// TwinCAT 3 PLC project lev_fsm
// ProgramVersion: 3.1.4023.0
// libraries:
//   Tc2_SerialCom, * (Beckhoff Automation GmbH)
//   Tc2_Standard, * (Beckhoff Automation GmbH)
//   Tc2_System, * (Beckhoff Automation GmbH)
//   Tc2_Utilities, * (Beckhoff Automation GmbH)
//   Tc3_Module, * (Beckhoff Automation GmbH)
// project tree:
//   DUTs/ E_FsmError.TcDUT (not stored), E_FsmState.TcDUT (not stored), mag_bus.TcDUT, ST_Event.TcDUT (not stored), sus_bus.TcDUT (not stored)
//   / PlcTask.TcTTO (not stored)
//   POUs/ getFmagnetic.TcPOU, getTrajectory.TcPOU (not stored), LevitationEqualizingController.TcPOU, MAIN.TcPOU (not stored), runIpcFsm.TcPOU (not stored)
//   POUs/nicht aufgerufen/ FiniteStateMachine.TcPOU, GenerateTrajectory.TcPOU (not stored), Trajectory.TcPOU, UpdateEventTimestampWithSystemTime.TcPOU

// ---- DUTs/mag_bus.TcDUT
TYPE mag_bus:
    STRUCT
        Fmat: ARRAY [0..143] OF LREAL;
        zmat: ARRAY [0..143] OF LREAL;
        invFmat: ARRAY [0..143] OF LREAL;
        F_grid: ARRAY [0..16383] OF LREAL;
        z_grid: ARRAY [0..16383] OF LREAL;
        i_grid: ARRAY [0..16383] OF LREAL;
    END_STRUCT
END_TYPE

// ---- POUs/getFmagnetic.TcPOU
FUNCTION getFmagnetic : LREAL
VAR_INPUT
    I: LREAL;
    z: LREAL;
END_VAR
VAR
    Fmag_tmp: LREAL;
    Fmag_tmp_0: LREAL;
    Fmag_tmp_1: LREAL;
    Fmag_tmp_2: LREAL;
    Fmag_tmp_3: LREAL;
    Fmag_tmp_4: LREAL;
END_VAR

(* MATLAB Function: '<Root>/getFmag' *)
(* MATLAB Function 'getFmag': '<S1>:1' *)
(* '<S1>:1:2' p00 =  -4.108e+05; *)
(* '<S1>:1:3' p10 =        3267; *)
(* '<S1>:1:4' p01 =   1.697e+05; *)
(* '<S1>:1:5' p20 =       61.45; *)
(* '<S1>:1:6' p11 =       -1147; *)
(* '<S1>:1:7' p02 =   -2.79e+04; *)
(* '<S1>:1:8' p30 =     -0.5002; *)
(* '<S1>:1:9' p21 =      -8.054; *)
(* '<S1>:1:10' p12 =       147.8; *)
(* '<S1>:1:11' p03 =        2282; *)
(* '<S1>:1:12' p40 =    -0.01962; *)
(* '<S1>:1:13' p31 =      0.1688; *)
(* '<S1>:1:14' p22 =      0.1559; *)
(* '<S1>:1:15' p13 =      -8.184; *)
(* '<S1>:1:16' p04 =      -92.92; *)
(* '<S1>:1:17' p50 =   0.0002649; *)
(* '<S1>:1:18' p41 =   -0.001089; *)
(* '<S1>:1:19' p32 =   -0.001289; *)
(* '<S1>:1:20' p23 =   -0.003046; *)
(* '<S1>:1:21' p14 =      0.1725; *)
(* '<S1>:1:22' p05 =       1.506; *)
(* '<S1>:1:23' Fmag = p00 + p10*I + p01*z + p20*I^2 + p11*I*z + p02*z^2 + p30*I^3 + p21*I^2*z + p12*I*z^2 + p03*z^3 + p40*I^4 + p31*I^3*z + p22*I^2*z^2 + p13*I*z^3 + p04*z^4 + p50*I^5 + p41*I^4*z + p32*I^3*z^2 + p23*I^2*z^3 + p14*I*z^4 + p05*z^5; *)
Fmag_tmp := EXPT(I, 3.0);
Fmag_tmp_0 := EXPT(z, 3.0);
Fmag_tmp_1 := EXPT(I, 4.0);
Fmag_tmp_2 := EXPT(z, 4.0);
Fmag_tmp_3 := I * I;
Fmag_tmp_4 := z * z;
getFmagnetic := ((((((((((((((((((((3267.0 * I) - 410800.0) + (169700.0 * z)) + (Fmag_tmp_3 * 61.45)) + ((-1147.0 * I) * z)) + (Fmag_tmp_4 * -27900.0)) + (-0.5002 * Fmag_tmp)) + ((Fmag_tmp_3 * -8.054) * z)) + ((147.8 * I) * Fmag_tmp_4)) + (2282.0 * Fmag_tmp_0)) + (-0.01962 * Fmag_tmp_1)) + ((0.1688 * Fmag_tmp) * z)) + ((Fmag_tmp_3 * 0.1559) * Fmag_tmp_4)) + ((-8.184 * I) * Fmag_tmp_0)) + (-92.92 * Fmag_tmp_2)) + (0.0002649 * EXPT(I, 5.0))) + ((-0.001089 * Fmag_tmp_1) * z)) + ((-0.001289 * Fmag_tmp) * Fmag_tmp_4)) + ((Fmag_tmp_3 * -0.003046) * Fmag_tmp_0)) + ((0.1725 * I) * Fmag_tmp_2)) + (1.506 * EXPT(z, 5.0));

END_FUNCTION

// ---- POUs/LevitationEqualizingController.TcPOU
FUNCTION_BLOCK LevitationEqualizingController
VAR_INPUT
	// Actual delta F value
	fActualdF : LREAL;
END_VAR

VAR
	// PID function block	
	fbPID : FB_BasicPID;
	// PID parameters
	fSetpointValue : LREAL;
	bReset : BOOL;
	fCtrlCycleTime : LREAL;
	fKp : LREAL;
	fTn : LREAL;
	fTv : LREAL;
	fTd : LREAL;
	// PID outputs	
	fCtrlOutput : LREAL;
	// Saturation parameter
	fdzMax : LREAL := 0.001;
	fdzMin : LREAL := -0.001;
END_VAR
VAR_OUTPUT
	// dz output vector
	fdz : ARRAY[1..4] OF LREAL;
	nErrorStatus : UINT;
END_VAR

fbPID(fSetpointValue := fSetpointValue,
	  fActualValue := fActualdF,
	  bReset := bReset,
	  fCtrlCycleTime := fCtrlCycleTime,
	  fKp := fKp,
	  fTn := fTn,
	  fTv := fTv,
	  fTd := fTd,
	  fCtrlOutput => fCtrlOutput, nErrorStatus => nErrorStatus);
	  
// Update the dz output vector
fdz[1] := -1/7900*fCtrlOutput; // TO DO : change it to lookup table function F_inv(F)
fdz[2] := 1/7900*fCtrlOutput;
fdz[3] := -1/7900*fCtrlOutput;
fdz[4] := 1/7900*fCtrlOutput;	  

// Saturate the dz output vector
IF fdz[1] > fdzMax THEN
	fdz[1] := fdzMax;
ELSIF fdz[1] < fdzMin THEN
	fdz[1] := fdzMin;
END_IF

IF fdz[2] > fdzMax THEN
	fdz[2] := fdzMax;
ELSIF fdz[2] < fdzMin THEN
	fdz[2] := fdzMin;
END_IF

IF fdz[3] > fdzMax THEN
	fdz[3] := fdzMax;
ELSIF fdz[3] < fdzMin THEN
	fdz[3] := fdzMin;
END_IF

IF fdz[4] > fdzMax THEN
	fdz[4] := fdzMax;
ELSIF fdz[4] < fdzMin THEN
	fdz[4] := fdzMin;
END_IF

METHOD FB_init : BOOL
VAR_INPUT
	bInitRetains : BOOL; // if TRUE, the retain variables are initialized (warm start / cold start)
	bInCopyCode : BOOL;  // if TRUE, the instance afterwards gets moved into the copy code (online change)
	fSetpointValue : LREAL;
	bReset : BOOL;
	fCtrlCycleTime : LREAL;
	fKp : LREAL;
	fTn : LREAL;
	fTv : LREAL;
	fTd : LREAL;
END_VAR
THIS^.fSetpointValue := fSetpointValue;
THIS^.bReset := bReset;
THIS^.fCtrlCycleTime := fCtrlCycleTime;
THIS^.fKp := fKp;
THIS^.fTn := fTn;
THIS^.fTv := fTv;
THIS^.fTd := fTd;
END_METHOD

END_FUNCTION_BLOCK

// ---- POUs/nicht aufgerufen/FiniteStateMachine.TcPOU
FUNCTION FiniteStateMachine : E_FsmState
VAR_INPUT
	eArgFsmState : E_FsmState;
END_VAR
VAR
END_VAR

CASE eArgFsmState OF
	//0
	E_FsmState.ERR:
		FiniteStateMachine := E_FsmState.ERR;
	//1
	E_FsmState.INIT:
		FiniteStateMachine := E_FsmState.INIT;
	//2
	E_FsmState.STAT:
		FiniteStateMachine := E_FsmState.STAT;
	//3
	E_FsmState.STAT_TR:
		FiniteStateMachine := E_FsmState.STAT_TR;
	//4
	E_FsmState.NOM_LEV:
		FiniteStateMachine := E_FsmState.NOM_LEV;
	//5
	E_FsmState.INTER_TR:
		FiniteStateMachine := E_FsmState.INTER_TR;
	//6
	E_FsmState.END_TR:
		FiniteStateMachine := E_FsmState.END_TR;
END_CASE

END_FUNCTION

// ---- POUs/nicht aufgerufen/Trajectory.TcPOU
FUNCTION_BLOCK Trajectory
VAR
	// Reference vector
	x_ref : ARRAY[1..3] OF REAL := [0.01, 0, 32.5]; // [z_nom, v_des, I_nom]
	// Nominal air gap
	z_nom : REAL := x_ref[1];
	// Desired vertical velocity at nominal state
	v_des : REAL := x_ref[2];
	// Nominal current
	I_nom: REAL := x_ref[3];
END_VAR
VAR CONSTANT
	Z_MAX : REAL := 0.025; // 25 mm
	Z_MIN : REAL := 0.002; // 2 mm
	I_MAX : REAL := 100; // 100 A
	I_MIN : REAL := 0; // 0 A
END_VAR

METHOD PUBLIC GenerateTrajectory

VAR_INPUT
	z_meas : REAL;
	v_meas : REAL;
	I_meas : REAL;
END_VAR
END_METHOD

END_FUNCTION_BLOCK

// ---- POUs/nicht aufgerufen/UpdateEventTimestampWithSystemTime.TcPOU
FUNCTION UpdateEventTimestampWithSystemTime
VAR_INPUT
	stEvent: REFERENCE TO ST_Event;
END_VAR
VAR
	fbGETSYSTEMTIME: GETSYSTEMTIME;
	stFileTime: T_FILETIME;
END_VAR

fbGETSYSTEMTIME(timeLoDW=> stFileTime.dwLowDateTime,
				timeHiDW=> stFileTime.dwHighDateTime);
stEvent.dtTimestamp := FILETIME_TO_DT(fileTime := stFileTime);

END_FUNCTION
